PROGRAM PRG_RestartPlc
VAR
END_VAR
VAR_INPUT
	CmdRestart 	: BOOL;
END_VAR

VAR
	RestartProcess : NT_Reboot;
	Trig_Restart	: R_TRIG;
	
END_VAR

Trig_Restart(CLK := CmdRestart);

RestartProcess
(
	NETID := '',
	START := Trig_Restart.Q,
	DELAY := 5,
	TMOUT := T#1S
);

END_PROGRAM

(* stored: Version 1.1.0.1, ProductVersion 3.1.4024.6
   POU PRG_RestartPlc: Id {a9da522d-bcf3-4058-af5e-42eb5ef1f88a}, SpecialFunc None *)
